PROGRAM PRG_LogHandlerManual
VAR
	
	stSystemTime			: TIMESTRUCT;
	sUTCTimeZone			: STRING(6);
	
	fbLogHandler			: LOGGER.FB_EventHandler;

	bLogData				: BOOL;
	sLogMessage				: T_LongSTRING;
	
	stEventDataUT				: LOGGER.ST_EventData;
	
	sResultMessage				: T_LongSTRING;
	
	bDone					: BOOL;
	bBufferOverflow			: BOOL;
END_VAR

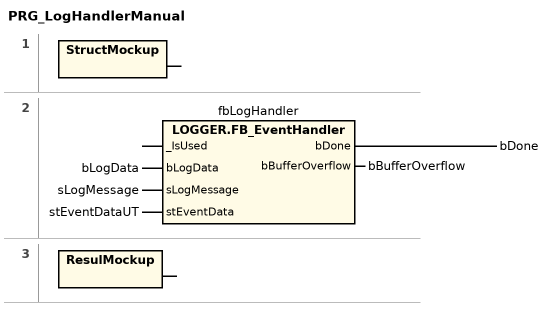
// NETWORK 1
StructMockup();

// NETWORK 2
fbLogHandler(
    bLogData := bLogData,
    sLogMessage := sLogMessage,
    stEventData := stEventDataUT,
    bBufferOverflow => bBufferOverflow); // LOGGER.FB_EventHandler
bDone := fbLogHandler.bDone;

// NETWORK 3
ResulMockup();

ACTION ResulMockup:
IF stEventDataUT.nImageByte < SIZEOF(sResultMessage) THEN
	MEMMOVE(ADR(sResultMessage), ADR(stEventDataUT.aDataLogImage), stEventDataUT.nImageByte);
END_IF
END_ACTION

ACTION StructMockup:

stEventDataUT.bEnable := TRUE;
stEventDataUT.sTimeStamp :=MID( F_SYSTEM_SystemTimeAsISO8601(stSystemTime, sUTCTimeZone ), 12, 12);

sLogMessage := '$01ST=53;$02CT=10;DS=GZDNP5JOA3IL;OG=3;XP=-50;YP=50;AP=-88;CS=06.2;SC=0070;QS=3;PN=1;$03
					$01ST=53;$02CT=10;DS=N7E1Y89UNK3O;OG=3;XP=-50;YP=-50;AP=-88;CS=06.2;SC=0070;QS=3;PN=2;$03
					$01ST=53;$02CT=10;DS=JHWJXYFNX9DS;OG=3;XP=50;YP=50;AP=-88;CS=06.2;SC=0070;QS=3;PN=3;$03
					$01ST=53;$02CT=10;DS=XGBEZLBV8A9I;OG=3;XP=50;YP=-50;AP=-88;CS=06.2;SC=0070;QS=3;PN=4;$03';
END_ACTION

END_PROGRAM

(* stored: Version 1.1.0.1
   POU PRG_LogHandlerManual: Id {8b4da0ab-55cf-415d-b8bc-1494441c783c}, SpecialFunc None
   Action ResulMockup: Id {8c8cd8da-3400-4252-ba12-807f6f8a7f1e}
   Action StructMockup: Id {2e2d3edf-0830-4130-b72d-13c360e6d388} *)
